// SIMATIC S7-200 project (STEP 7-Micro/WIN), CPU 224XP REL 02.01

SYMBOL_TABLE USUARIO1
MARCHA           I0.0
FC               I0.1
C_FOTOELECTRICA  I0.2
PARO             I0.3
CINTA_1          Q0.0
LED_CINTA_1      Q0.1
BAJADA_PISTON    Q0.2
SUBIDA_PISTON    Q0.3
MOTOR_TALADRO    Q0.4
LED_PISTON       Q0.5
LED_PARO         Q0.6
END_SYMBOL_TABLE

SYMBOL_TABLE Símbolos S7-200
Primer_ciclo_ON  SM0.1    // ON sólo en el primer ciclo
END_SYMBOL_TABLE

ORGANIZATION_BLOCK PRINCIPAL:OB1
TITLE=COMENTARIOS DEL PROGRAMA
BEGIN
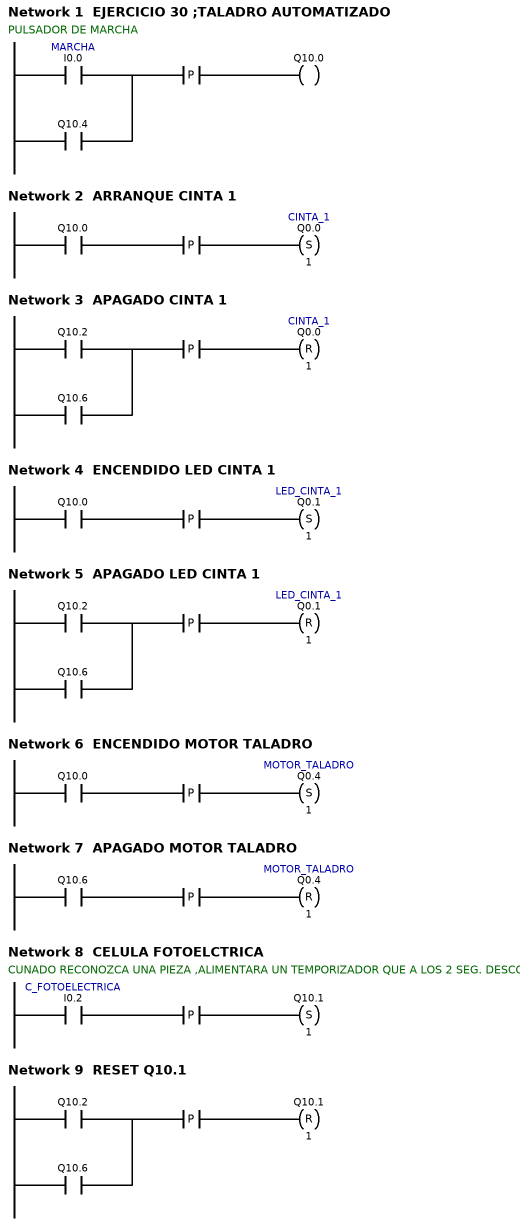
Network 1 // EJERCICIO 30 ;TALADRO AUTOMATIZADO
// PULSADOR DE MARCHA
LD     MARCHA:I0.0
O      Q10.4
EU
=      Q10.0
Network 2 // ARRANQUE CINTA 1 
LD     Q10.0
EU
S      CINTA_1:Q0.0, 1
Network 3 // APAGADO CINTA 1
LD     Q10.2
O      Q10.6
EU
R      CINTA_1:Q0.0, 1
Network 4 // ENCENDIDO LED CINTA 1
LD     Q10.0
EU
S      LED_CINTA_1:Q0.1, 1
Network 5 // APAGADO LED CINTA 1
LD     Q10.2
O      Q10.6
EU
R      LED_CINTA_1:Q0.1, 1
Network 6 // ENCENDIDO MOTOR TALADRO
LD     Q10.0
EU
S      MOTOR_TALADRO:Q0.4, 1
Network 7 // APAGADO MOTOR TALADRO
LD     Q10.6
EU
R      MOTOR_TALADRO:Q0.4, 1
Network 8 // CELULA FOTOELCTRICA
// CUNADO RECONOZCA UNA PIEZA ,ALIMENTARA UN TEMPORIZADOR QUE A LOS 2 SEG. DESCONECTA LA CINTA 1 Y CONECTA LA BAJADA DEL PISTON.
LD     C_FOTOELECTRICA:I0.2
EU
S      Q10.1, 1
Network 9 // RESET Q10.1 
LD     Q10.2
O      Q10.6
EU
R      Q10.1, 1
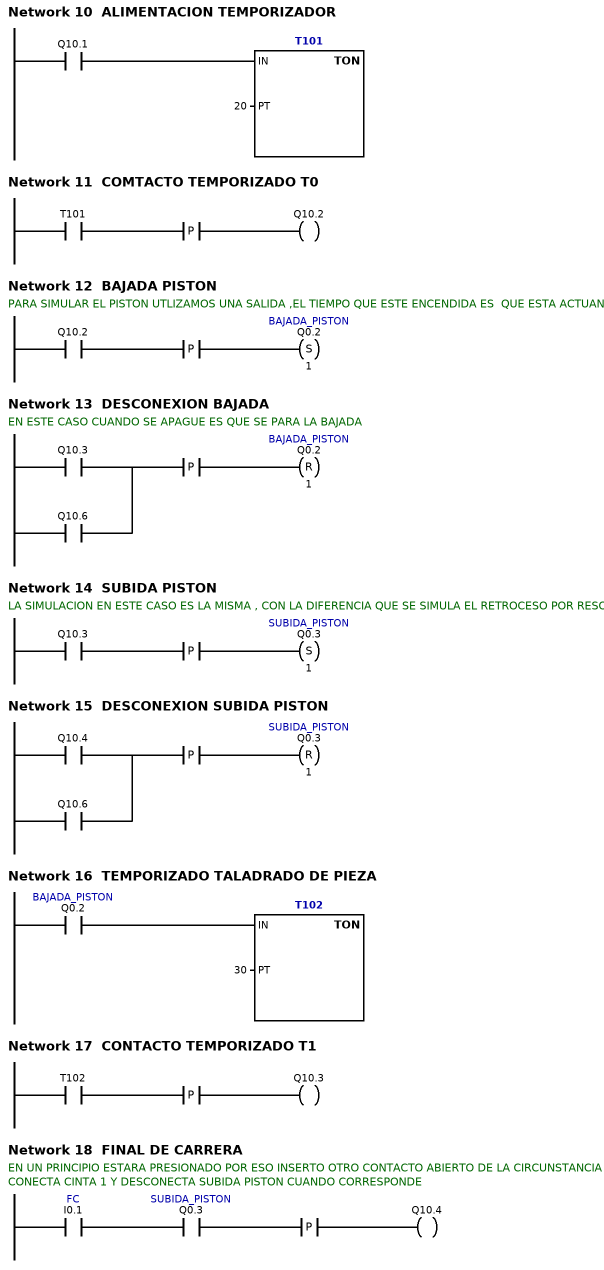
Network 10 // ALIMENTACION TEMPORIZADOR
LD     Q10.1
TON    T101, 20
Network 11 // COMTACTO TEMPORIZADO T0
LD     T101
EU
=      Q10.2
Network 12 // BAJADA PISTON 
// PARA SIMULAR EL PISTON UTLIZAMOS UNA SALIDA ,EL TIEMPO QUE ESTE ENCENDIDA ES  QUE ESTA ACTUANDO SOBRE LA BAJADA 
LD     Q10.2
EU
S      BAJADA_PISTON:Q0.2, 1
Network 13 // DESCONEXION BAJADA 
// EN ESTE CASO CUANDO SE APAGUE ES QUE SE PARA LA BAJADA 
LD     Q10.3
O      Q10.6
EU
R      BAJADA_PISTON:Q0.2, 1
Network 14 // SUBIDA PISTON
// LA SIMULACION EN ESTE CASO ES LA MISMA , CON LA DIFERENCIA QUE SE SIMULA EL RETROCESO POR RESORTE 
LD     Q10.3
EU
S      SUBIDA_PISTON:Q0.3, 1
Network 15 // DESCONEXION SUBIDA PISTON
LD     Q10.4
O      Q10.6
EU
R      SUBIDA_PISTON:Q0.3, 1
Network 16 // TEMPORIZADO TALADRADO DE PIEZA
LD     BAJADA_PISTON:Q0.2
TON    T102, 30
Network 17 // CONTACTO TEMPORIZADO T1
LD     T102
EU
=      Q10.3
Network 18 // FINAL DE CARRERA
// EN UN PRINCIPIO ESTARA PRESIONADO POR ESO INSERTO OTRO CONTACTO ABIERTO DE LA CIRCUNSTANCIA QUE PRECEDE A ESTA EJECUCION ,QUE ES LA SUBIDA DEL PISTON Y ACTO SEGUIDO CONECTA CINTA 1 Y DESCONECTA SUBIDA PISTON CUANDO CORRESPONDE
LD     FC:I0.1
A      SUBIDA_PISTON:Q0.3
EU
=      Q10.4
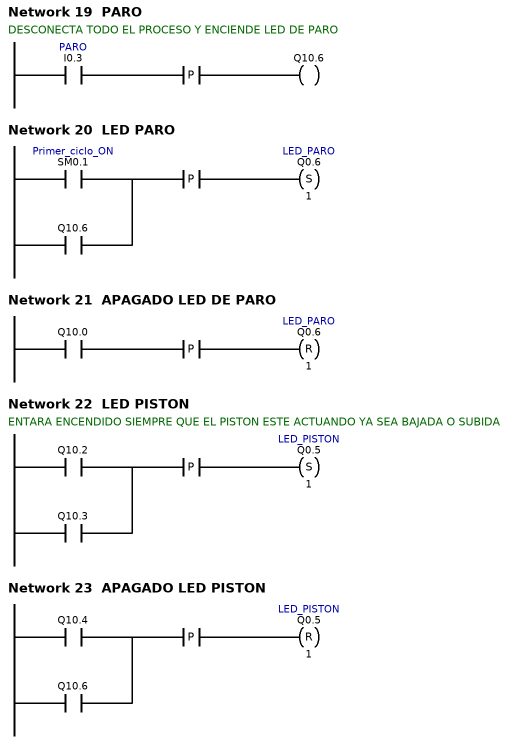
Network 19 // PARO
// DESCONECTA TODO EL PROCESO Y ENCIENDE LED DE PARO
LD     PARO:I0.3
EU
=      Q10.6
Network 20 // LED PARO
LD     Primer_ciclo_ON:SM0.1
O      Q10.6
EU
S      LED_PARO:Q0.6, 1
Network 21 // APAGADO LED DE PARO
LD     Q10.0
EU
R      LED_PARO:Q0.6, 1
Network 22 // LED PISTON
// ENTARA ENCENDIDO SIEMPRE QUE EL PISTON ESTE ACTUANDO YA SEA BAJADA O SUBIDA
LD     Q10.2
O      Q10.3
EU
S      LED_PISTON:Q0.5, 1
Network 23 // APAGADO LED PISTON
LD     Q10.4
O      Q10.6
EU
R      LED_PISTON:Q0.5, 1
END_ORGANIZATION_BLOCK
